(* CODESYS project GuardClausesExport.export

Project tree, tasks and I/O mapping:
  program Main [ST]: DoSomething, LogError
*)

// Main
PROGRAM Main
VAR
	ConditionA : BOOL;
	ConditionB : BOOL;
	ConditionC : BOOL;
END_VAR


// Instead of this -->
IF ConditionA THEN
    IF ConditionB THEN
        IF NOT ConditionC THEN
            DoSomething();
		ELSE
			LogError('ConditionC was true');
        END_IF
	ELSE
		LogError('ConditionB was false');
    END_IF
ELSE
	LogError('ConditionA was false');
END_IF


//----------------------------------------------------------------------------+

// Try this -->
IF NOT ConditionA THEN 
	LogError('ConditionA was false');
	RETURN; 
END_IF

IF NOT ConditionB THEN
	LogError('ConditionB was false');	
 	RETURN; 
END_IF

IF ConditionC THEN
	LogError('ConditionC was true'); 
	RETURN; 
END_IF

DoSomething();

METHOD PRIVATE DoSomething : BOOL
VAR_INPUT
END_VAR
END_METHOD

METHOD PUBLIC LogError
VAR_INPUT
	ErrorMessage : STRING;
END_VAR
END_METHOD

END_PROGRAM
